FUNCTION_BLOCK SPLIT_AD_INTO_AW (* this Function splits the 2 AW (WORD) adapters from a AD (DWORD) *)
  (* Standard: 61499-2; Description: Copyright (c) 2026 Meisterschulen am Ostbahnhof SPDX-License-Identifier: EPL-2.0 *)
  (* Version 1.0, 2026-05-16, Franz Höpfinger, Meisterschulen am Ostbahnhof, initial API and implementation and/or initial documentation *)
  PACKAGE adapter::splitting;
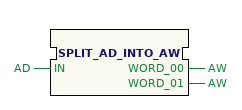
  SOCKETS
    IN : adapter::types::unidirectional::AD; (* DWORD Input *)
  END_SOCKETS
  PLUGS
    WORD_00 : adapter::types::unidirectional::AW; (* Word 0 *)
    WORD_01 : adapter::types::unidirectional::AW; (* Word 1 *)
  END_PLUGS
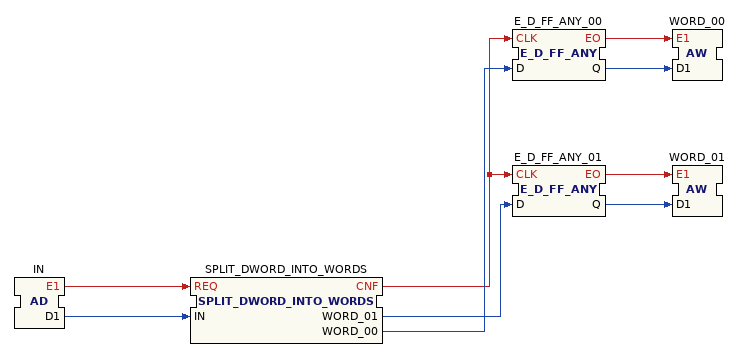
  FBS
    E_D_FF_ANY_00 : iec61499::events::E_D_FF_ANY;
    E_D_FF_ANY_01 : iec61499::events::E_D_FF_ANY;
    SPLIT_DWORD_INTO_WORDS : eclipse4diac::utils::splitting::SPLIT_DWORD_INTO_WORDS;
  END_FBS
  EVENT_CONNECTIONS
    IN.E1 TO SPLIT_DWORD_INTO_WORDS.REQ;
    SPLIT_DWORD_INTO_WORDS.CNF TO E_D_FF_ANY_00.CLK;
    SPLIT_DWORD_INTO_WORDS.CNF TO E_D_FF_ANY_01.CLK;
    E_D_FF_ANY_00.EO TO WORD_00.E1;
    E_D_FF_ANY_01.EO TO WORD_01.E1;
  END_CONNECTIONS
  DATA_CONNECTIONS
    IN.D1 TO SPLIT_DWORD_INTO_WORDS.IN;
    SPLIT_DWORD_INTO_WORDS.WORD_01 TO E_D_FF_ANY_01.D;
    SPLIT_DWORD_INTO_WORDS.WORD_00 TO E_D_FF_ANY_00.D;
    E_D_FF_ANY_00.Q TO WORD_00.D1;
    E_D_FF_ANY_01.Q TO WORD_01.D1;
  END_CONNECTIONS
END_FUNCTION_BLOCK
